FUNCTION_BLOCK TcAxis_DMC_Tc3_Direct_Motion_Control IMPLEMENTS itfAxis
VAR_INPUT
	Axis 				: Tc3_Direct_Motion_control.AXIS_REF();
END_VAR
//VAR_OUTPUT
//END_VAR
VAR
END_VAR

END_FUNCTION_BLOCK

(* stored: Version 1.1.0.1, ProductVersion 3.1.4024.12
   POU TcAxis_DMC_Tc3_Direct_Motion_Control: Id {2f6e3521-f867-48d7-93bf-b8218196dd59}, SpecialFunc None *)
